(* IEC 61131-3 sources: process-and-packaging-plant/codesys/level-tank, 4 files *)

(* ---- GVL_Level.st ---- *)
{attribute 'qualified_only'}
VAR_GLOBAL
	Level_PV : REAL := 50.0; // Process variable (measured level, 0-100%)
	Level_SP : REAL := 50.0; // Setpoint
	Kp : REAL := 2.0; // Proportional Gain (starting)
	Ki : REAL := 0.1; // Integral Gain (starting)
	Kd : REAL := 0; // Derivative Gain (initially zero)
	Controller_Output : REAL := 50; // PID Output, 0-100%
	Pump_Enable : BOOL; // Final Control Element
	Mode_Auto : BOOL := TRUE; // TRUE = PID, FALSE = Manual
	Prev_Mode_Auto : BOOL;
	Manual_Output : REAL := 0.0; // Manual Output value
	High_Alarm : BOOL;
	Low_Alarm : BOOL;
	High_Alarm_Trip : BOOL; // Trip for interlock
	Sim_Current : REAL; // Simulated pump current
	Overcurrent_Alarm : BOOL;
	Overcurrent_Threshold : REAL := 8.0; // Amps
	Outflow_Disturbance : REAL := 20.0; // Load Disturbance
	ScanTime : REAL := 0.1; // Scan time in seconds

	// For P-only Control
	Error : REAL;
    Prev_Error : REAL;
	P_Term : REAL;

	// For Integral and Anti-Windup
	I_Term : REAL;
	Integral : REAL;
	Output_Saturated : BOOL;
	Tf : REAL := 0.5; // Ideally 5-10x ScanTime as a rule of thumb

	// For Derivative and 1st Order Low Pass Filter
	D_Term : REAL;
	D_Raw : REAL;
	D_Filtered : REAL;
	Alpha : REAL;
	Prev_PV : REAL;

	// For Interlock LD
	Manual_Run : BOOL;
	ResetTrip : BOOL;

	// For random noise generation
    RandSeed : DWORD := 12345;   // any non-zero initial value
	Noise : REAL;

	// For Tank Simulation with Interlock
	Effective_Output : REAL;
END_VAR

(* ---- PLC_PRG_Alarms.st ---- *)
// High alarm with hysteresis (5% deadband)
// This is to avoid spillage, overflow, environmental hazards, contact with electrical equipment
IF GVL_Level.Level_PV > 90.0 THEN
	GVL_Level.High_Alarm := TRUE;
ELSIF GVL_Level.Level_PV < 85.0 THEN
	GVL_Level.High_Alarm := FALSE;
END_IF

// Low alarm with hysteresis
// This is to avoid motor overheating, cavitation, impeller damage, seal failure
IF GVL_Level.Level_PV < 10.0 THEN
	GVL_Level.Low_Alarm := TRUE;
ELSIF GVL_Level.Level_PV > 15.0 THEN
	GVL_Level.Low_Alarm := FALSE;
END_IF

// Hysteresis is used to prevent chatter

// High alarm trip (latched)
IF GVL_Level.High_Alarm THEN
    GVL_Level.High_Alarm_Trip := TRUE;
END_IF

(* ---- PLC_PRG_PID.st ---- *)
(* Our goal is to compute the manipulated variable (MV) for the level control loop using a
   discrete-time PID controller with anti-windup and bumpless transfer.

Controller Equation in continuous time is
 u(t) = Kp * e(t)  +  Ki * ∫e(t)dt  +  Kd * de(t)/dt
 where u(t) is Controller_Output (MV), e(t) is Error (setpoint Level_SP - process variable Level_PV), Kp is proportional gain, Ki is integral gain, Kd is derivative gain

 Level_PV is measured tank level (0-100%), Level_SP is desired tank level, Controller_Output (MV) is pump speed/valve position (0-100%)

 We implement controller equation in time domain because that's what PLC can handle, it dosen't need the entire process (which CLTF offers)
 CLTF is for analysis and Kp pre-tuning (calculating offset, closed loop time constant, damping), not for implementation

The PID reads PV and SP, computes error, and outputs MV.
The process (mock tank or Factory I/O scene) receives MV and changes PV.

Servo Test keeps disturbance (outflow) constant and step changes in SP (eg: 40 to 60%) to measure tracking response, especially rise time, overshoot, settling time
Regulatory Test keeps SP constant and step changes disturbance (eg: 50 to 70%) to measure disturbance rejection

Both tests are performed in the mock simulation before Factory I/O.
The tuning log records results from both.

After changing MV, the transient response is observed (changes in Servo and Regulatory related variables), measured in CODESYS watch window or Ignition trends.
rise time (time to reach 90% of final value), overshoot (peak value above SP in %), settling time (time to stay within 2% of SP), steady-state offset*)

// 1 - Proportional-only Control

GVL_Level.Error := GVL_Level.Level_SP - GVL_Level.Level_PV; // Error
GVL_Level.P_Term := GVL_Level.Kp * GVL_Level.Error; // Proportional Term

// 2 - Integral term with anti-windup (conditional integration)
// Only integrate if output is not saturated in the direction of the error
// Anti-windup prevents the integral from growing and causing overshoot after output saturates (eg, during startup or large steps)
(* INTEGRAL: Rectangular/Euler/Left Riemann Sum Approximation
     Continuous: I = ∫e(t)dt
     Discrete:   Integral := Integral + (Error * dt)
     Assumed constant error over each scan cycle. Good for small dt (100 ms). Error is O(dt).
	 Trapezoidal Rule is more accurate but more expensive to implement and unnecessary for small dt *)

GVL_Level.Output_Saturated := (GVL_Level.Controller_Output >= 100.0 AND GVL_Level.Error > 0.0) OR (GVL_Level.Controller_Output <= 0.0 AND GVL_Level.Error < 0.0);

IF NOT GVL_Level.Output_Saturated THEN
	GVL_Level.Integral := GVL_Level.Integral + (GVL_Level.Error * GVL_Level.ScanTime);
END_IF

GVL_Level.I_Term := GVL_Level.Ki * GVL_Level.Integral;

// 3 - Derivative Term with 1st order Filter
(* DERIVATIVE: Backward Difference Approximation
  Continuous: D = de(t)/dt
  Discrete:   D_term := Kd * (Level_PV - Previous_PV) / dt
  Note that derivative is taken on (Level_PV - Prev_PV) over (Error - Prev_Error) to avoid "derivative kick" when SP changes abruptly.
  Also note that derivatives amplify sensor noise which is why PI is preferred for Level Tanks and real PLCs apply a filter to D, not noticeable in Mock Tank but there in Factory I/O *)

 GVL_Level.D_Raw := (GVL_Level.Kd*(GVL_Level.Level_PV - GVL_Level.Prev_PV)) / GVL_Level.ScanTime ;
 GVL_Level.Prev_PV := GVL_Level.Level_PV;

  (* A 1st order Low Pass Filter is used on D, using the Backward Euler Approximation, the industry standard
  Continuous: D(s) = Kd * s / (1 + Tf*s) * PV(s)
  Discrete:   D_filtered[k] = alpha * D_filtered[k-1] + (1-alpha) * D_raw[k]
  where:      alpha = Tf / (Tf + dt)
  Backward Euler is stable for any dt and Tf, only has one multiply-add per scan, avoids phase lead, has sufficient accuracy
  Forward Euler needs dt < 2Tf to be stable, Matched Pole-Zero uses exp(), hence both are rare in industry. Tustin (bilinear) is too complex and introduces phase lead near Nyquist frequency, but occassionally used in industry. *)

  GVL_Level.Alpha := GVL_Level.Tf / (GVL_Level.Tf + GVL_Level.ScanTime);
  GVL_Level.D_Filtered := (GVL_Level.Alpha * GVL_Level.D_Filtered) + ((1.0 - GVL_Level.Alpha) * GVL_Level.D_Raw);
  GVL_Level.D_Term := GVL_Level.D_Filtered;

// 4 - Controller Output (MV)

IF GVL_Level.Mode_Auto THEN
	// Bumpless Transfer (manual to auto) - Initialize integral so that output matches manual value
	IF NOT GVL_Level.Prev_Mode_Auto THEN
		IF  GVL_Level.Ki <> 0.0 THEN
			GVL_Level.Integral := (GVL_Level.Manual_Output - GVL_Level.P_Term - GVL_Level.D_Term)/(GVL_Level.Ki);
		END_IF
	END_IF
	GVL_Level.Controller_Output := GVL_Level.P_Term + GVL_Level.I_Term + GVL_Level.D_Term;
ELSE
	// Manual Mode : MV directly set by operator
	GVL_Level.Controller_Output := GVL_Level.Manual_Output;
END_IF

GVL_Level.Prev_Mode_Auto := GVL_Level.Mode_Auto;

// 5 - Clamp Output to 0-100%
// Physical limits of pump/valve

IF GVL_Level.Controller_Output > 100.0 THEN
	GVL_Level.Controller_Output := 100.0;
ELSIF GVL_Level.Controller_Output < 0.0 THEN
	GVL_Level.Controller_Output := 0.0;
END_IF

(* ---- PLC_PRG_TankSim.st ---- *)
// Mock Tank Physics
// A 1st order level model with inflow from the pump and outflow as the disturbance
// Level changes based on (inflow - outflow) * dt
// Controller Output is 0-100%, representing pump speed/valve position

GVL_Level.Level_PV := GVL_Level.Level_PV + (GVL_Level.Controller_Output - GVL_Level.Outflow_Disturbance) * GVL_Level.ScanTime * 0.01;
// The 0.01 value is arbitrary to keep level response ata  realistic range given output is 0-100
// The key is that Level_PV integrates the difference between inflow and outflow

// Clamp Level to 0-100%

IF GVL_Level.Level_PV > 100.0 THEN
	GVL_Level.Level_PV := 100.0;
ELSIF GVL_Level.Level_PV < 0.0 THEN
	GVL_Level.Level_PV := 0.0;
END_IF
